// TIA Portal V19 export
VAR_GLOBAL   // PLC tag table "03_SAFETY_SINAMICS_A02"
   Cassetta1_OP_StsIn AT %I710.0 : "udt_LDrvSafe_typeSinaSTlg30Status";
   Cassetta1_OP_CtrlOut AT %Q710.0 : "udt_LDrvSafe_typeSinaSTlg30Control";
   Cassetta1_MOT_StsIn AT %I720.0 : "udt_LDrvSafe_typeSinaSTlg30Status";
   Cassetta1_MOT_CtrlOut AT %Q720.0 : "udt_LDrvSafe_typeSinaSTlg30Control";
   Cassetta2_OP_StsIn AT %I730.0 : "udt_LDrvSafe_typeSinaSTlg30Control";
   Cassetta2_OP_CtrlOut AT %Q730.0 : "udt_LDrvSafe_typeSinaSTlg30Control";
   Cassetta2_MOT_StsIn AT %I740.0 : "udt_LDrvSafe_typeSinaSTlg30Control";
   Cassetta2_MOT_CtrlOut AT %Q740.0 : "udt_LDrvSafe_typeSinaSTlg30Control";
   Cassetta3_OP_StsIn AT %I750.0 : "udt_LDrvSafe_typeSinaSTlg30Control";
   Cassetta3_OP_CtrlOut AT %Q750.0 : "udt_LDrvSafe_typeSinaSTlg30Control";
   Cassetta3_MOT_StsIn AT %I760.0 : "udt_LDrvSafe_typeSinaSTlg30Control";
   Cassetta3_MOT_CtrlOut AT %Q760.0 : "udt_LDrvSafe_typeSinaSTlg30Control";
   Rollfomer_StsIn AT %I276.0 : "udt_LDrvSafe_typeSinaSTlg30Control";
   Rollfomer_CtrlOut AT %Q276.0 : "udt_LDrvSafe_typeSinaSTlg30Control";
   FAK_Pusher_StsIn AT %I648.0 : "udt_LDrvSafe_typeSinaSTlg30Control";
   FAK_Pusher_CtrlOut AT %Q648.0 : "udt_LDrvSafe_typeSinaSTlg30Control";
   Carriage_StsIn AT %I282.0 : "udt_LDrvSafe_typeSinaSTlg30Control";
   Carriage_CtrlOut AT %Q282.0 : "udt_LDrvSafe_typeSinaSTlg30Control";
   AccRolls1_StsIn AT %I608.0 : "udt_LDrvSafe_typeSinaSTlg30Control";
   AccRolls1_CtrlOut AT %Q608.0 : "udt_LDrvSafe_typeSinaSTlg30Control";
   AccRolls2_StsIn AT %I618.0 : "udt_LDrvSafe_typeSinaSTlg30Control";
   AccRolls2_CtrlOut AT %Q618.0 : "udt_LDrvSafe_typeSinaSTlg30Control";
   AccRolls3_StsIn AT %I628.0 : "udt_LDrvSafe_typeSinaSTlg30Control";
   AccRolls3_CtrlOut AT %Q628.0 : "udt_LDrvSafe_typeSinaSTlg30Control";
END_VAR
